% RSLogix 500 project PV8M.RSS, saved by version 8.30.00.16 %
PROJECT "PV8M"    % processor: Bul.1763 MicroLogix 1100 Series B %

PROGRAM FILES
  LAD 2   64 rungs

DATA FILES
  O0 OUTPUT  5 elements
  I1 INPUT  7 elements
  S2 STATUS  66 elements
  B3 BINARY  6 elements
  T4 TIMER  9 elements
  C5 COUNTER  1 elements
  R6 CONTROL  1 elements
  N7 INTEGER  11 elements
  F8 FLOAT  1 elements

LADDER 2
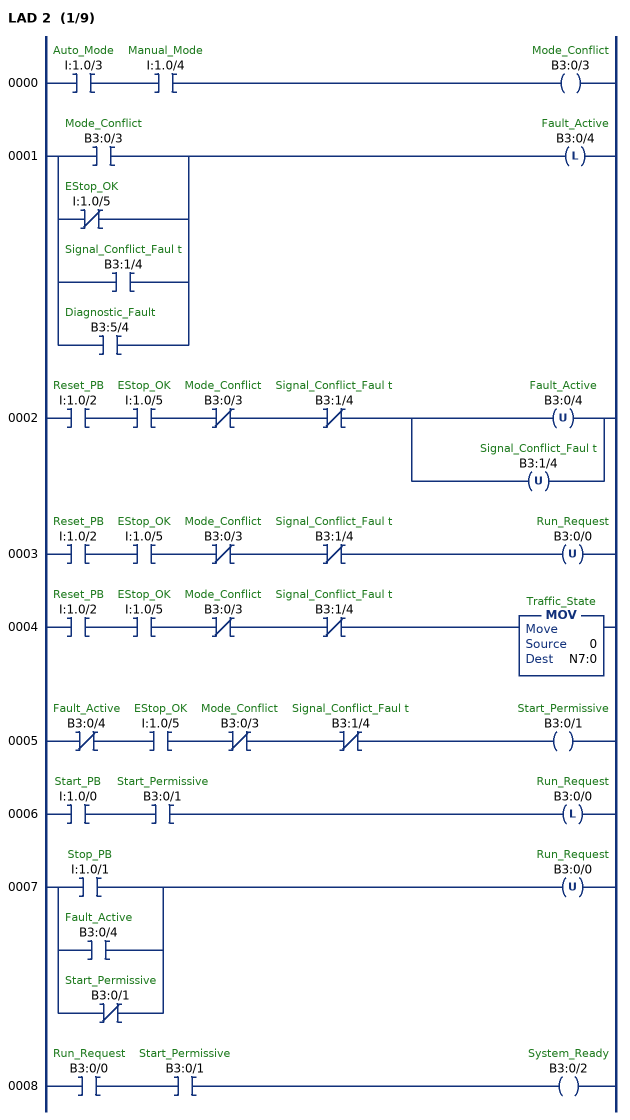
% Rung: 0 %
SOR XIC I:1.0/3 XIC I:1.0/4 OTE B3:0/3 EOR
%   I:1.0/3  "Auto_Mode" %
%   I:1.0/4  "Manual_Mode" %
%   B3:0/3  "Mode_Conflict" %
% Rung: 1 %
SOR BST XIC B3:0/3 NXB BST XIO I:1.0/5 NXB BST XIC B3:1/4 NXB XIC B3:5/4 BND BND BND OTL B3:0/4 EOR
%   B3:0/3  "Mode_Conflict" %
%   I:1.0/5  "EStop_OK" %
%   B3:1/4  "Signal_Conflict_Faul t" %
%   B3:5/4  "Diagnostic_Fault" %
%   B3:0/4  "Fault_Active" %
% Rung: 2 %
SOR XIC I:1.0/2 XIC I:1.0/5 XIO B3:0/3 XIO B3:1/4 BST OTU B3:0/4 NXB OTU B3:1/4 BND EOR
%   I:1.0/2  "Reset_PB" %
%   I:1.0/5  "EStop_OK" %
%   B3:0/3  "Mode_Conflict" %
%   B3:1/4  "Signal_Conflict_Faul t" %
%   B3:0/4  "Fault_Active" %
% Rung: 3 %
SOR XIC I:1.0/2 XIC I:1.0/5 XIO B3:0/3 XIO B3:1/4 OTU B3:0/0 EOR
%   I:1.0/2  "Reset_PB" %
%   I:1.0/5  "EStop_OK" %
%   B3:0/3  "Mode_Conflict" %
%   B3:1/4  "Signal_Conflict_Faul t" %
%   B3:0/0  "Run_Request" %
% Rung: 4 %
SOR XIC I:1.0/2 XIC I:1.0/5 XIO B3:0/3 XIO B3:1/4 MOV 0 N7:0 EOR
%   I:1.0/2  "Reset_PB" %
%   I:1.0/5  "EStop_OK" %
%   B3:0/3  "Mode_Conflict" %
%   B3:1/4  "Signal_Conflict_Faul t" %
%   N7:0  "Traffic_State" %
% Rung: 5 %
SOR XIO B3:0/4 XIC I:1.0/5 XIO B3:0/3 XIO B3:1/4 OTE B3:0/1 EOR
%   B3:0/4  "Fault_Active" %
%   I:1.0/5  "EStop_OK" %
%   B3:0/3  "Mode_Conflict" %
%   B3:1/4  "Signal_Conflict_Faul t" %
%   B3:0/1  "Start_Permissive" %
% Rung: 6 %
SOR XIC I:1.0/0 XIC B3:0/1 OTL B3:0/0 EOR
%   I:1.0/0  "Start_PB" %
%   B3:0/1  "Start_Permissive" %
%   B3:0/0  "Run_Request" %
% Rung: 7 %
SOR BST XIC I:1.0/1 NXB BST XIC B3:0/4 NXB XIO B3:0/1 BND BND OTU B3:0/0 EOR
%   I:1.0/1  "Stop_PB" %
%   B3:0/4  "Fault_Active" %
%   B3:0/1  "Start_Permissive" %
%   B3:0/0  "Run_Request" %
% Rung: 8 %
SOR XIC B3:0/0 XIC B3:0/1 OTE B3:0/2 EOR
%   B3:0/0  "Run_Request" %
%   B3:0/1  "Start_Permissive" %
%   B3:0/2  "System_Ready" %

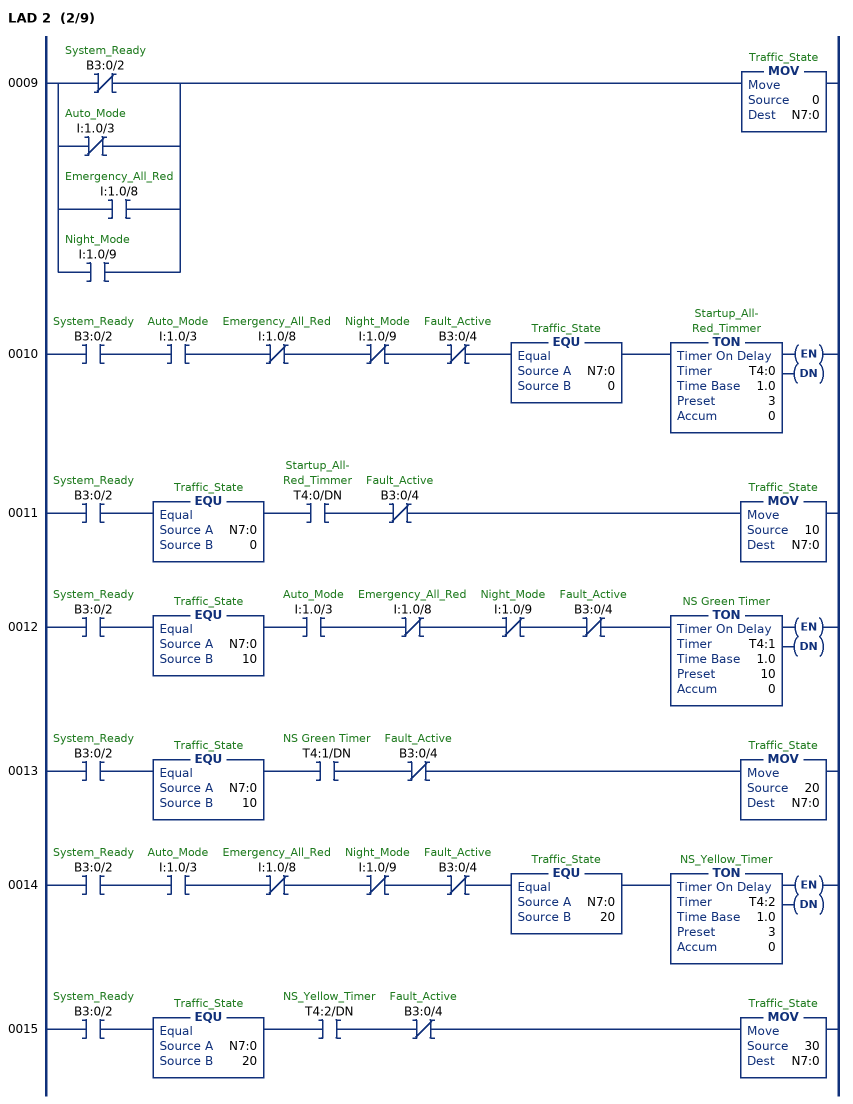
% Rung: 9 %
SOR BST XIO B3:0/2 NXB BST XIO I:1.0/3 NXB BST XIC I:1.0/8 NXB XIC I:1.0/9 BND BND BND MOV 0 N7:0 EOR
%   B3:0/2  "System_Ready" %
%   I:1.0/3  "Auto_Mode" %
%   I:1.0/8  "Emergency_All_Red" %
%   I:1.0/9  "Night_Mode" %
%   N7:0  "Traffic_State" %
% Rung: 10 %
SOR XIC B3:0/2 XIC I:1.0/3 XIO I:1.0/8 XIO I:1.0/9 XIO B3:0/4 EQU N7:0 0 TON T4:0 1.0 3 0 EOR
%   B3:0/2  "System_Ready" %
%   I:1.0/3  "Auto_Mode" %
%   I:1.0/8  "Emergency_All_Red" %
%   I:1.0/9  "Night_Mode" %
%   B3:0/4  "Fault_Active" %
%   N7:0  "Traffic_State" %
%   T4:0  "Startup_All- Red_Timmer" %
% Rung: 11 %
SOR XIC B3:0/2 EQU N7:0 0 XIC T4:0/DN XIO B3:0/4 MOV 10 N7:0 EOR
%   B3:0/2  "System_Ready" %
%   N7:0  "Traffic_State" %
%   T4:0  "Startup_All- Red_Timmer" %
%   B3:0/4  "Fault_Active" %
% Rung: 12 %
SOR XIC B3:0/2 EQU N7:0 10 XIC I:1.0/3 XIO I:1.0/8 XIO I:1.0/9 XIO B3:0/4 TON T4:1 1.0 10 0 EOR
%   B3:0/2  "System_Ready" %
%   N7:0  "Traffic_State" %
%   I:1.0/3  "Auto_Mode" %
%   I:1.0/8  "Emergency_All_Red" %
%   I:1.0/9  "Night_Mode" %
%   B3:0/4  "Fault_Active" %
%   T4:1  "NS Green Timer" %
% Rung: 13 %
SOR XIC B3:0/2 EQU N7:0 10 XIC T4:1/DN XIO B3:0/4 MOV 20 N7:0 EOR
%   B3:0/2  "System_Ready" %
%   N7:0  "Traffic_State" %
%   T4:1  "NS Green Timer" %
%   B3:0/4  "Fault_Active" %
% Rung: 14 %
SOR XIC B3:0/2 XIC I:1.0/3 XIO I:1.0/8 XIO I:1.0/9 XIO B3:0/4 EQU N7:0 20 TON T4:2 1.0 3 0 EOR
%   B3:0/2  "System_Ready" %
%   I:1.0/3  "Auto_Mode" %
%   I:1.0/8  "Emergency_All_Red" %
%   I:1.0/9  "Night_Mode" %
%   B3:0/4  "Fault_Active" %
%   N7:0  "Traffic_State" %
%   T4:2  "NS_Yellow_Timer" %
% Rung: 15 %
SOR XIC B3:0/2 EQU N7:0 20 XIC T4:2/DN XIO B3:0/4 MOV 30 N7:0 EOR
%   B3:0/2  "System_Ready" %
%   N7:0  "Traffic_State" %
%   T4:2  "NS_Yellow_Timer" %
%   B3:0/4  "Fault_Active" %

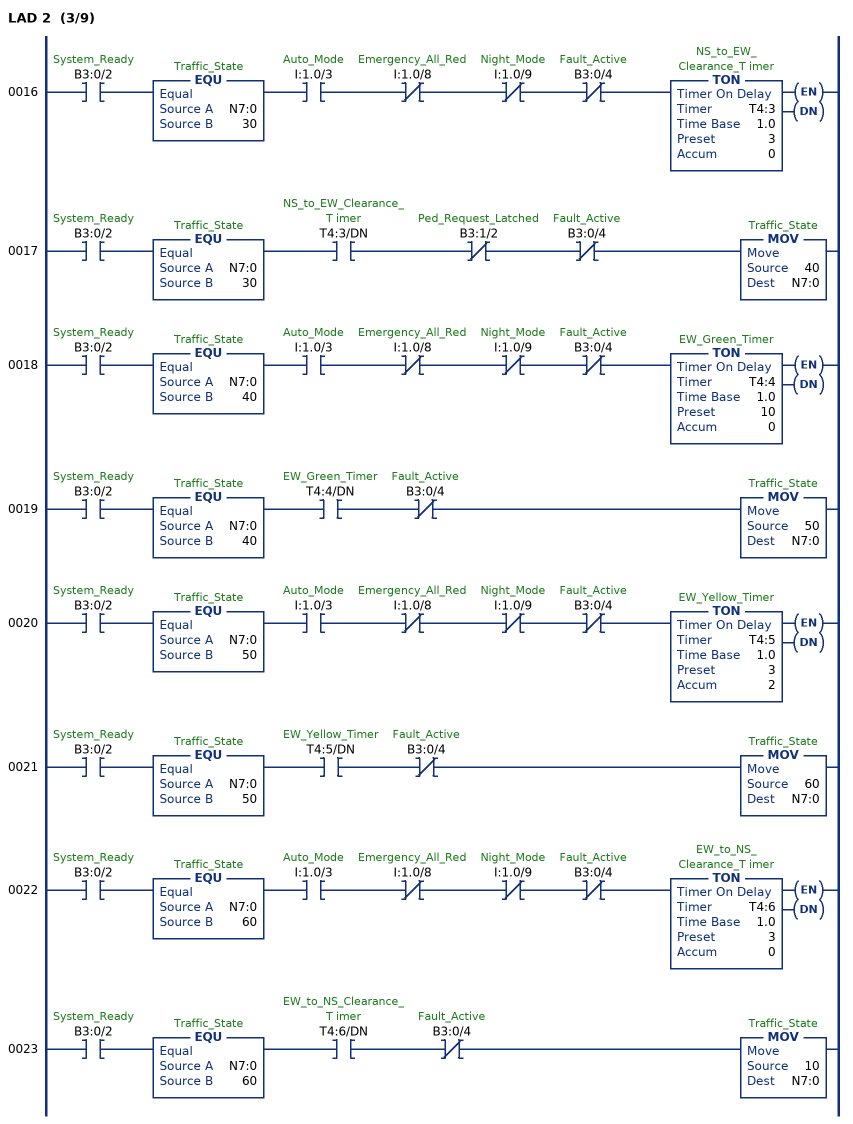
% Rung: 16 %
SOR XIC B3:0/2 EQU N7:0 30 XIC I:1.0/3 XIO I:1.0/8 XIO I:1.0/9 XIO B3:0/4 TON T4:3 1.0 3 0 EOR
%   B3:0/2  "System_Ready" %
%   N7:0  "Traffic_State" %
%   I:1.0/3  "Auto_Mode" %
%   I:1.0/8  "Emergency_All_Red" %
%   I:1.0/9  "Night_Mode" %
%   B3:0/4  "Fault_Active" %
%   T4:3  "NS_to_EW_Clearance_T imer" %
% Rung: 17 %
SOR XIC B3:0/2 EQU N7:0 30 XIC T4:3/DN XIO B3:1/2 XIO B3:0/4 MOV 40 N7:0 EOR
%   B3:0/2  "System_Ready" %
%   N7:0  "Traffic_State" %
%   T4:3  "NS_to_EW_Clearance_T imer" %
%   B3:1/2  "Ped_Request_Latched" %
%   B3:0/4  "Fault_Active" %
% Rung: 18 %
SOR XIC B3:0/2 EQU N7:0 40 XIC I:1.0/3 XIO I:1.0/8 XIO I:1.0/9 XIO B3:0/4 TON T4:4 1.0 10 0 EOR
%   B3:0/2  "System_Ready" %
%   N7:0  "Traffic_State" %
%   I:1.0/3  "Auto_Mode" %
%   I:1.0/8  "Emergency_All_Red" %
%   I:1.0/9  "Night_Mode" %
%   B3:0/4  "Fault_Active" %
%   T4:4  "EW_Green_Timer" %
% Rung: 19 %
SOR XIC B3:0/2 EQU N7:0 40 XIC T4:4/DN XIO B3:0/4 MOV 50 N7:0 EOR
%   B3:0/2  "System_Ready" %
%   N7:0  "Traffic_State" %
%   T4:4  "EW_Green_Timer" %
%   B3:0/4  "Fault_Active" %
% Rung: 20 %
SOR XIC B3:0/2 EQU N7:0 50 XIC I:1.0/3 XIO I:1.0/8 XIO I:1.0/9 XIO B3:0/4 TON T4:5 1.0 3 2 EOR
%   B3:0/2  "System_Ready" %
%   N7:0  "Traffic_State" %
%   I:1.0/3  "Auto_Mode" %
%   I:1.0/8  "Emergency_All_Red" %
%   I:1.0/9  "Night_Mode" %
%   B3:0/4  "Fault_Active" %
%   T4:5  "EW_Yellow_Timer" %
% Rung: 21 %
SOR XIC B3:0/2 EQU N7:0 50 XIC T4:5/DN XIO B3:0/4 MOV 60 N7:0 EOR
%   B3:0/2  "System_Ready" %
%   N7:0  "Traffic_State" %
%   T4:5  "EW_Yellow_Timer" %
%   B3:0/4  "Fault_Active" %
% Rung: 22 %
SOR XIC B3:0/2 EQU N7:0 60 XIC I:1.0/3 XIO I:1.0/8 XIO I:1.0/9 XIO B3:0/4 TON T4:6 1.0 3 0 EOR
%   B3:0/2  "System_Ready" %
%   N7:0  "Traffic_State" %
%   I:1.0/3  "Auto_Mode" %
%   I:1.0/8  "Emergency_All_Red" %
%   I:1.0/9  "Night_Mode" %
%   B3:0/4  "Fault_Active" %
%   T4:6  "EW_to_NS_Clearance_T imer" %
% Rung: 23 %
SOR XIC B3:0/2 EQU N7:0 60 XIC T4:6/DN XIO B3:0/4 MOV 10 N7:0 EOR
%   B3:0/2  "System_Ready" %
%   N7:0  "Traffic_State" %
%   T4:6  "EW_to_NS_Clearance_T imer" %
%   B3:0/4  "Fault_Active" %

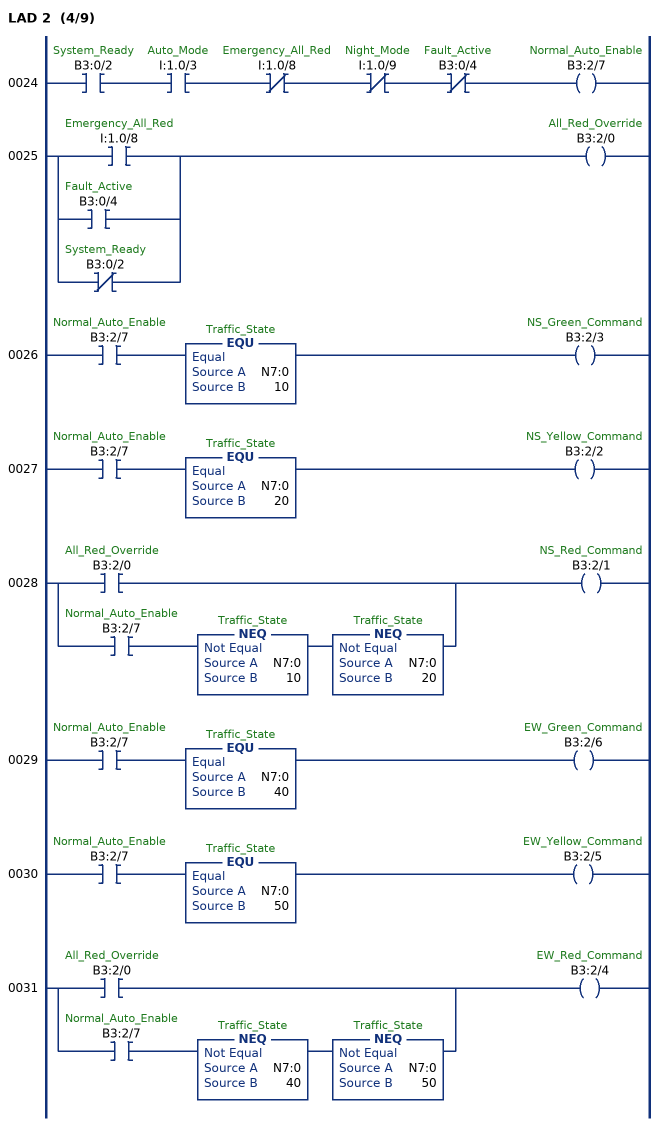
% Rung: 24 %
SOR XIC B3:0/2 XIC I:1.0/3 XIO I:1.0/8 XIO I:1.0/9 XIO B3:0/4 OTE B3:2/7 EOR
%   B3:0/2  "System_Ready" %
%   I:1.0/3  "Auto_Mode" %
%   I:1.0/8  "Emergency_All_Red" %
%   I:1.0/9  "Night_Mode" %
%   B3:0/4  "Fault_Active" %
%   B3:2/7  "Normal_Auto_Enable" %
% Rung: 25 %
SOR BST XIC I:1.0/8 NXB BST XIC B3:0/4 NXB XIO B3:0/2 BND BND OTE B3:2/0 EOR
%   I:1.0/8  "Emergency_All_Red" %
%   B3:0/4  "Fault_Active" %
%   B3:0/2  "System_Ready" %
%   B3:2/0  "All_Red_Override" %
% Rung: 26 %
SOR XIC B3:2/7 EQU N7:0 10 OTE B3:2/3 EOR
%   B3:2/7  "Normal_Auto_Enable" %
%   N7:0  "Traffic_State" %
%   B3:2/3  "NS_Green_Command" %
% Rung: 27 %
SOR XIC B3:2/7 EQU N7:0 20 OTE B3:2/2 EOR
%   B3:2/7  "Normal_Auto_Enable" %
%   N7:0  "Traffic_State" %
%   B3:2/2  "NS_Yellow_Command" %
% Rung: 28 %
SOR BST XIC B3:2/0 NXB XIC B3:2/7 NEQ N7:0 10 NEQ N7:0 20 BND OTE B3:2/1 EOR
%   B3:2/0  "All_Red_Override" %
%   B3:2/7  "Normal_Auto_Enable" %
%   N7:0  "Traffic_State" %
%   B3:2/1  "NS_Red_Command" %
% Rung: 29 %
SOR XIC B3:2/7 EQU N7:0 40 OTE B3:2/6 EOR
%   B3:2/7  "Normal_Auto_Enable" %
%   N7:0  "Traffic_State" %
%   B3:2/6  "EW_Green_Command" %
% Rung: 30 %
SOR XIC B3:2/7 EQU N7:0 50 OTE B3:2/5 EOR
%   B3:2/7  "Normal_Auto_Enable" %
%   N7:0  "Traffic_State" %
%   B3:2/5  "EW_Yellow_Command" %
% Rung: 31 %
SOR BST XIC B3:2/0 NXB XIC B3:2/7 NEQ N7:0 40 NEQ N7:0 50 BND OTE B3:2/4 EOR
%   B3:2/0  "All_Red_Override" %
%   B3:2/7  "Normal_Auto_Enable" %
%   N7:0  "Traffic_State" %
%   B3:2/4  "EW_Red_Command" %

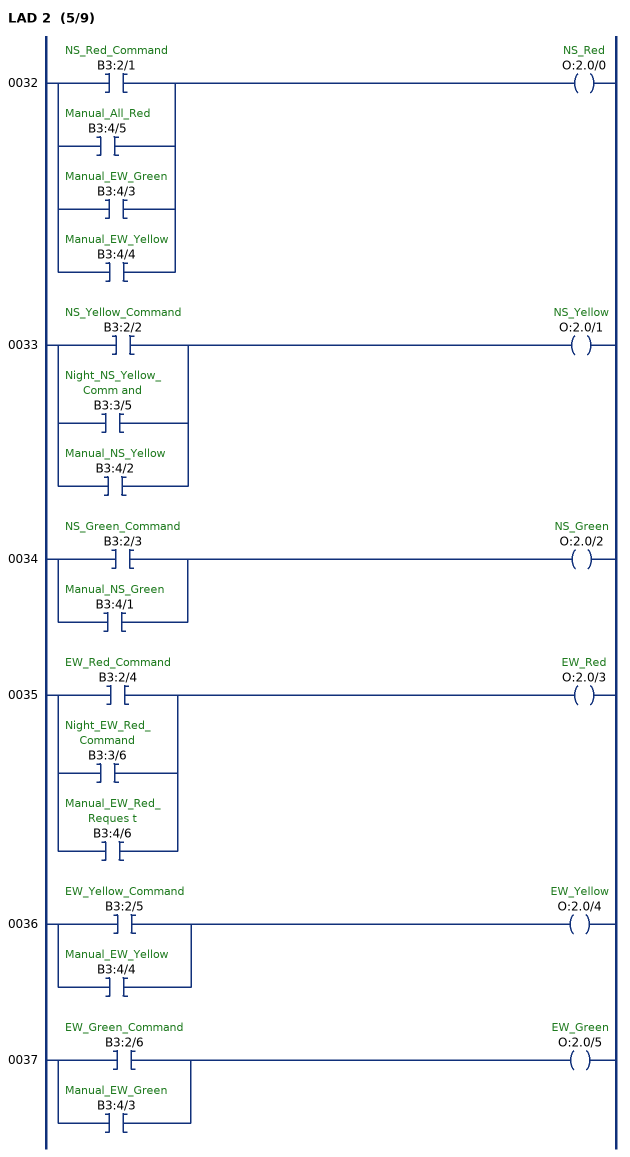
% Rung: 32 %
SOR BST XIC B3:2/1 NXB BST XIC B3:4/5 NXB BST XIC B3:4/3 NXB XIC B3:4/4 BND BND BND OTE O:2.0/0 EOR
%   B3:2/1  "NS_Red_Command" %
%   B3:4/5  "Manual_All_Red" %
%   B3:4/3  "Manual_EW_Green" %
%   B3:4/4  "Manual_EW_Yellow" %
%   O:2.0/0  "NS_Red" %
% Rung: 33 %
SOR BST XIC B3:2/2 NXB BST XIC B3:3/5 NXB XIC B3:4/2 BND BND OTE O:2.0/1 EOR
%   B3:2/2  "NS_Yellow_Command" %
%   B3:3/5  "Night_NS_Yellow_Comm and" %
%   B3:4/2  "Manual_NS_Yellow" %
%   O:2.0/1  "NS_Yellow" %
% Rung: 34 %
SOR BST XIC B3:2/3 NXB XIC B3:4/1 BND OTE O:2.0/2 EOR
%   B3:2/3  "NS_Green_Command" %
%   B3:4/1  "Manual_NS_Green" %
%   O:2.0/2  "NS_Green" %
% Rung: 35 %
SOR BST XIC B3:2/4 NXB BST XIC B3:3/6 NXB XIC B3:4/6 BND BND OTE O:2.0/3 EOR
%   B3:2/4  "EW_Red_Command" %
%   B3:3/6  "Night_EW_Red_Command" %
%   B3:4/6  "Manual_EW_Red_Reques t" %
%   O:2.0/3  "EW_Red" %
% Rung: 36 %
SOR BST XIC B3:2/5 NXB XIC B3:4/4 BND OTE O:2.0/4 EOR
%   B3:2/5  "EW_Yellow_Command" %
%   B3:4/4  "Manual_EW_Yellow" %
%   O:2.0/4  "EW_Yellow" %
% Rung: 37 %
SOR BST XIC B3:2/6 NXB XIC B3:4/3 BND OTE O:2.0/5 EOR
%   B3:2/6  "EW_Green_Command" %
%   B3:4/3  "Manual_EW_Green" %
%   O:2.0/5  "EW_Green" %

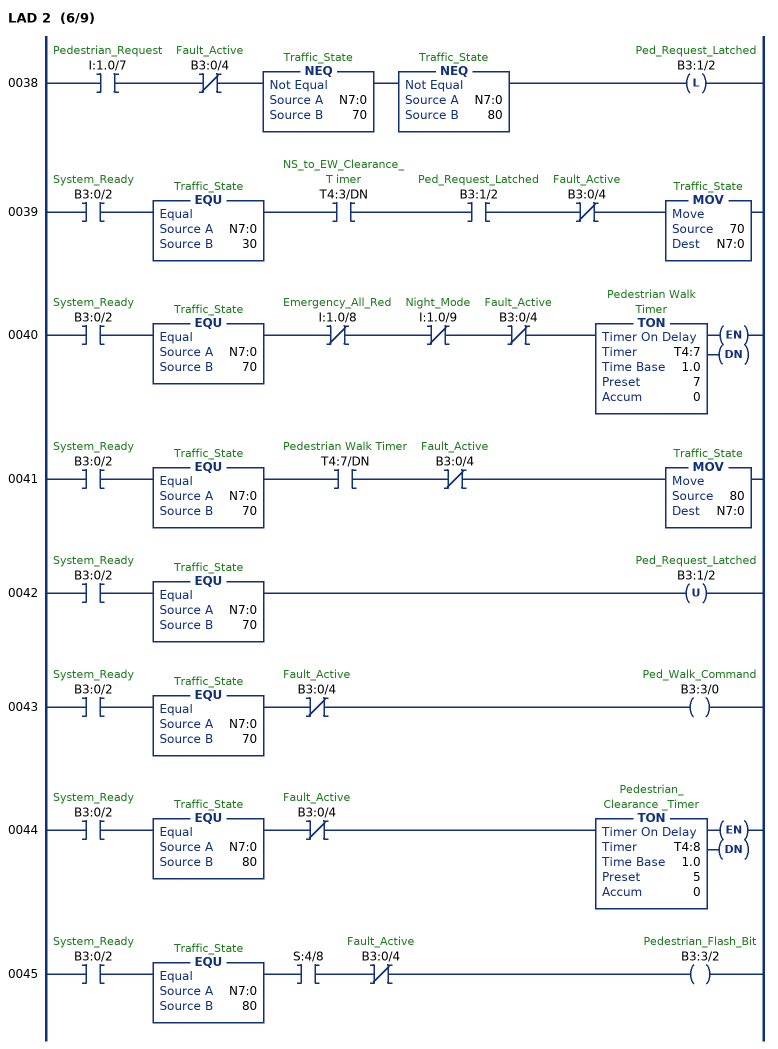
% Rung: 38 %
SOR XIC I:1.0/7 XIO B3:0/4 NEQ N7:0 70 NEQ N7:0 80 OTL B3:1/2 EOR
%   I:1.0/7  "Pedestrian_Request" %
%   B3:0/4  "Fault_Active" %
%   N7:0  "Traffic_State" %
%   B3:1/2  "Ped_Request_Latched" %
% Rung: 39 %
SOR XIC B3:0/2 EQU N7:0 30 XIC T4:3/DN XIC B3:1/2 XIO B3:0/4 MOV 70 N7:0 EOR
%   B3:0/2  "System_Ready" %
%   N7:0  "Traffic_State" %
%   T4:3  "NS_to_EW_Clearance_T imer" %
%   B3:1/2  "Ped_Request_Latched" %
%   B3:0/4  "Fault_Active" %
% Rung: 40 %
SOR XIC B3:0/2 EQU N7:0 70 XIO I:1.0/8 XIO I:1.0/9 XIO B3:0/4 TON T4:7 1.0 7 0 EOR
%   B3:0/2  "System_Ready" %
%   N7:0  "Traffic_State" %
%   I:1.0/8  "Emergency_All_Red" %
%   I:1.0/9  "Night_Mode" %
%   B3:0/4  "Fault_Active" %
%   T4:7  "Pedestrian Walk Timer" %
% Rung: 41 %
SOR XIC B3:0/2 EQU N7:0 70 XIC T4:7/DN XIO B3:0/4 MOV 80 N7:0 EOR
%   B3:0/2  "System_Ready" %
%   N7:0  "Traffic_State" %
%   T4:7  "Pedestrian Walk Timer" %
%   B3:0/4  "Fault_Active" %
% Rung: 42 %
SOR XIC B3:0/2 EQU N7:0 70 OTU B3:1/2 EOR
%   B3:0/2  "System_Ready" %
%   N7:0  "Traffic_State" %
%   B3:1/2  "Ped_Request_Latched" %
% Rung: 43 %
SOR XIC B3:0/2 EQU N7:0 70 XIO B3:0/4 OTE B3:3/0 EOR
%   B3:0/2  "System_Ready" %
%   N7:0  "Traffic_State" %
%   B3:0/4  "Fault_Active" %
%   B3:3/0  "Ped_Walk_Command" %
% Rung: 44 %
SOR XIC B3:0/2 EQU N7:0 80 XIO B3:0/4 TON T4:8 1.0 5 0 EOR
%   B3:0/2  "System_Ready" %
%   N7:0  "Traffic_State" %
%   B3:0/4  "Fault_Active" %
%   T4:8  "Pedestrian_Clearance _Timer" %
% Rung: 45 %
SOR XIC B3:0/2 EQU N7:0 80 XIC S:4/8 XIO B3:0/4 OTE B3:3/2 EOR
%   B3:0/2  "System_Ready" %
%   N7:0  "Traffic_State" %
%   B3:0/4  "Fault_Active" %
%   B3:3/2  "Pedestrian_Flash_Bit" %

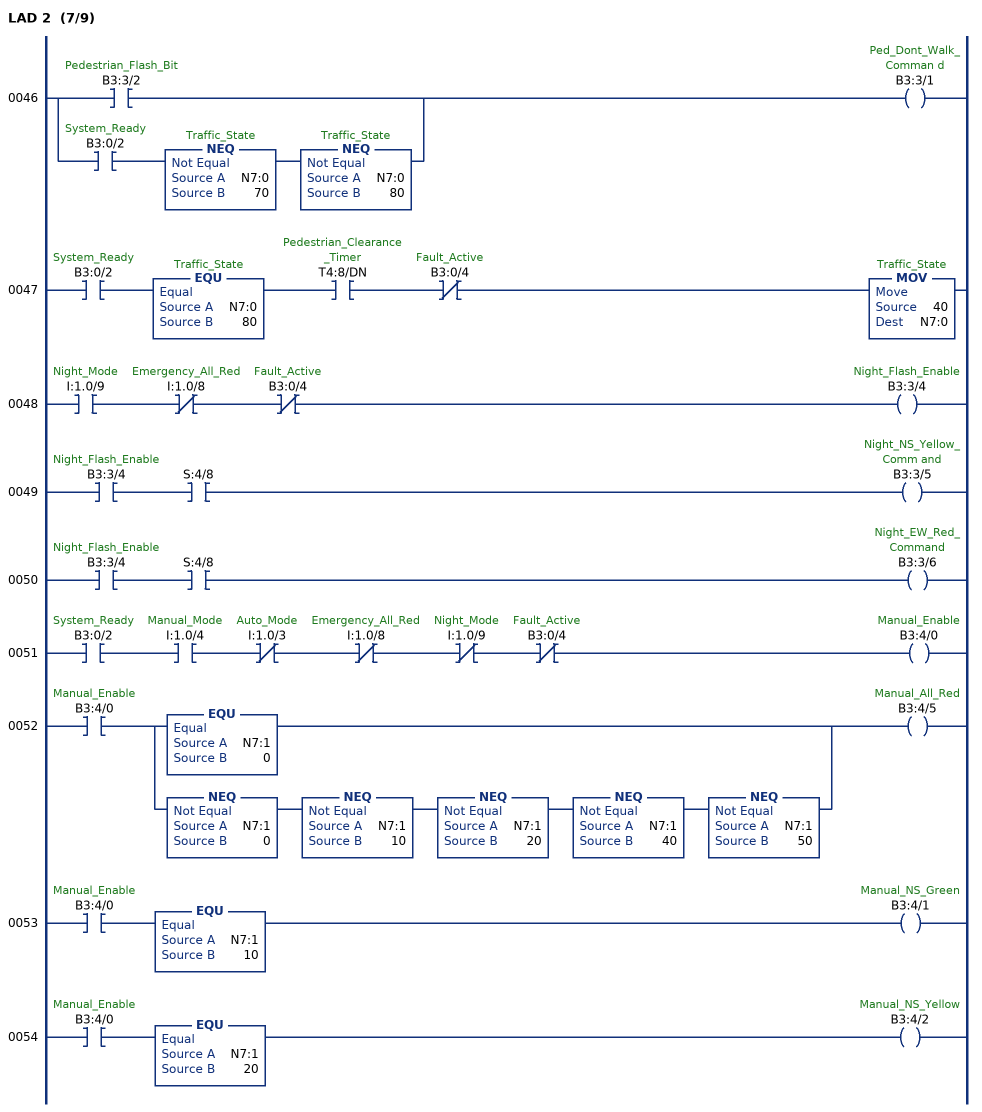
% Rung: 46 %
SOR BST XIC B3:3/2 NXB XIC B3:0/2 NEQ N7:0 70 NEQ N7:0 80 BND OTE B3:3/1 EOR
%   B3:3/2  "Pedestrian_Flash_Bit" %
%   B3:0/2  "System_Ready" %
%   N7:0  "Traffic_State" %
%   B3:3/1  "Ped_Dont_Walk_Comman d" %
% Rung: 47 %
SOR XIC B3:0/2 EQU N7:0 80 XIC T4:8/DN XIO B3:0/4 MOV 40 N7:0 EOR
%   B3:0/2  "System_Ready" %
%   N7:0  "Traffic_State" %
%   T4:8  "Pedestrian_Clearance _Timer" %
%   B3:0/4  "Fault_Active" %
% Rung: 48 %
SOR XIC I:1.0/9 XIO I:1.0/8 XIO B3:0/4 OTE B3:3/4 EOR
%   I:1.0/9  "Night_Mode" %
%   I:1.0/8  "Emergency_All_Red" %
%   B3:0/4  "Fault_Active" %
%   B3:3/4  "Night_Flash_Enable" %
% Rung: 49 %
SOR XIC B3:3/4 XIC S:4/8 OTE B3:3/5 EOR
%   B3:3/4  "Night_Flash_Enable" %
%   B3:3/5  "Night_NS_Yellow_Comm and" %
% Rung: 50 %
SOR XIC B3:3/4 XIC S:4/8 OTE B3:3/6 EOR
%   B3:3/4  "Night_Flash_Enable" %
%   B3:3/6  "Night_EW_Red_Command" %
% Rung: 51 %
SOR XIC B3:0/2 XIC I:1.0/4 XIO I:1.0/3 XIO I:1.0/8 XIO I:1.0/9 XIO B3:0/4 OTE B3:4/0 EOR
%   B3:0/2  "System_Ready" %
%   I:1.0/4  "Manual_Mode" %
%   I:1.0/3  "Auto_Mode" %
%   I:1.0/8  "Emergency_All_Red" %
%   I:1.0/9  "Night_Mode" %
%   B3:0/4  "Fault_Active" %
%   B3:4/0  "Manual_Enable" %
% Rung: 52 %
SOR XIC B3:4/0 BST EQU N7:1 0 NXB NEQ N7:1 0 NEQ N7:1 10 NEQ N7:1 20 NEQ N7:1 40 NEQ N7:1 50 BND OTE B3:4/5 EOR
%   B3:4/0  "Manual_Enable" %
%   B3:4/5  "Manual_All_Red" %
% Rung: 53 %
SOR XIC B3:4/0 EQU N7:1 10 OTE B3:4/1 EOR
%   B3:4/0  "Manual_Enable" %
%   B3:4/1  "Manual_NS_Green" %
% Rung: 54 %
SOR XIC B3:4/0 EQU N7:1 20 OTE B3:4/2 EOR
%   B3:4/0  "Manual_Enable" %
%   B3:4/2  "Manual_NS_Yellow" %

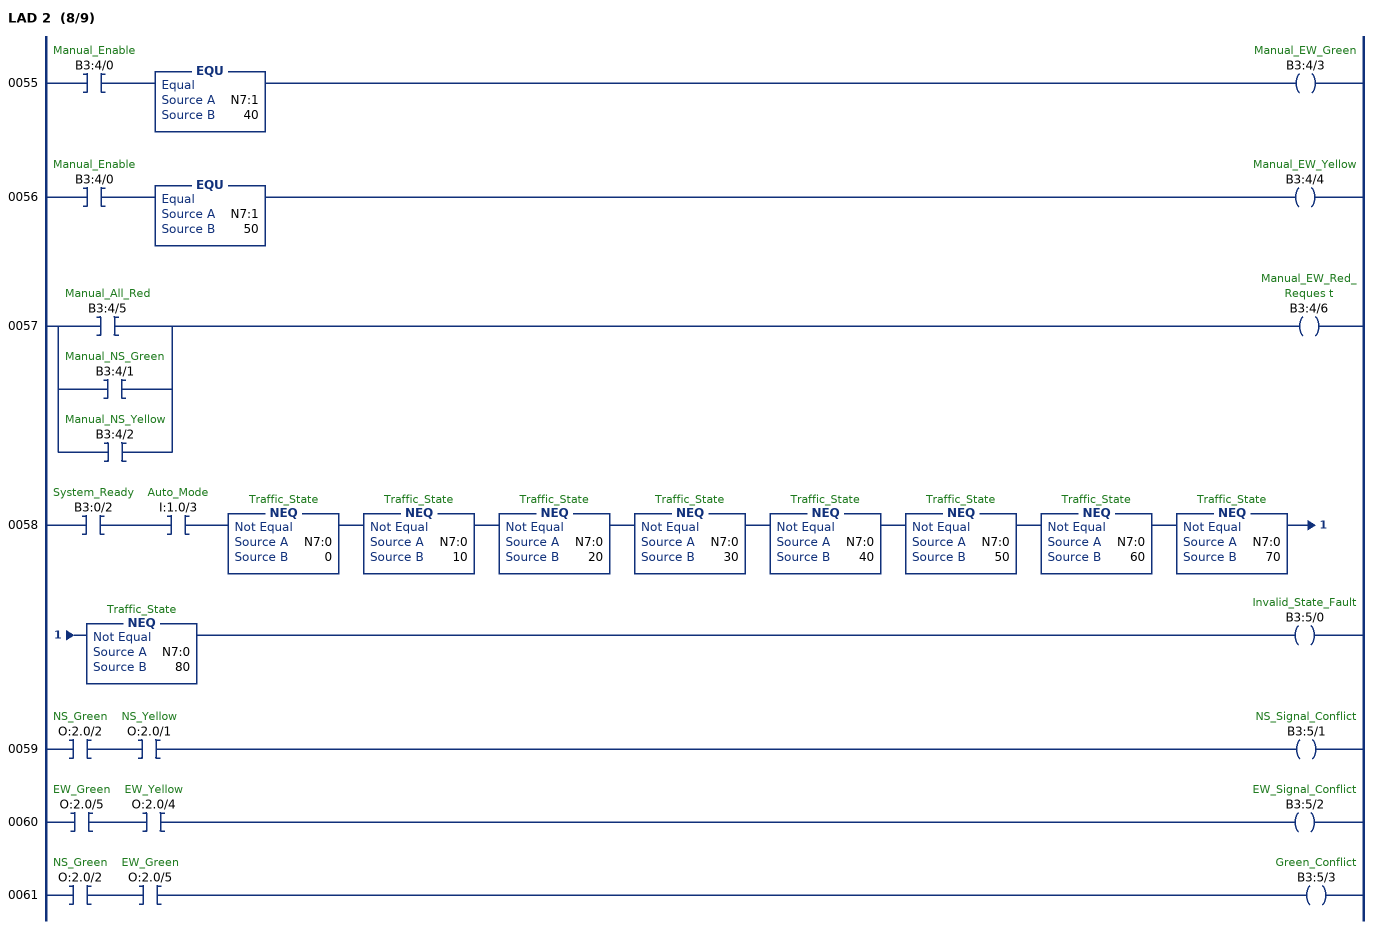
% Rung: 55 %
SOR XIC B3:4/0 EQU N7:1 40 OTE B3:4/3 EOR
%   B3:4/0  "Manual_Enable" %
%   B3:4/3  "Manual_EW_Green" %
% Rung: 56 %
SOR XIC B3:4/0 EQU N7:1 50 OTE B3:4/4 EOR
%   B3:4/0  "Manual_Enable" %
%   B3:4/4  "Manual_EW_Yellow" %
% Rung: 57 %
SOR BST XIC B3:4/5 NXB BST XIC B3:4/1 NXB XIC B3:4/2 BND BND OTE B3:4/6 EOR
%   B3:4/5  "Manual_All_Red" %
%   B3:4/1  "Manual_NS_Green" %
%   B3:4/2  "Manual_NS_Yellow" %
%   B3:4/6  "Manual_EW_Red_Reques t" %
% Rung: 58 %
SOR XIC B3:0/2 XIC I:1.0/3 NEQ N7:0 0 NEQ N7:0 10 NEQ N7:0 20 NEQ N7:0 30 NEQ N7:0 40 NEQ N7:0 50 NEQ N7:0 60 NEQ N7:0 70 NEQ N7:0 80 OTE B3:5/0 EOR
%   B3:0/2  "System_Ready" %
%   I:1.0/3  "Auto_Mode" %
%   N7:0  "Traffic_State" %
%   B3:5/0  "Invalid_State_Fault" %
% Rung: 59 %
SOR XIC O:2.0/2 XIC O:2.0/1 OTE B3:5/1 EOR
%   O:2.0/2  "NS_Green" %
%   O:2.0/1  "NS_Yellow" %
%   B3:5/1  "NS_Signal_Conflict" %
% Rung: 60 %
SOR XIC O:2.0/5 XIC O:2.0/4 OTE B3:5/2 EOR
%   O:2.0/5  "EW_Green" %
%   O:2.0/4  "EW_Yellow" %
%   B3:5/2  "EW_Signal_Conflict" %
% Rung: 61 %
SOR XIC O:2.0/2 XIC O:2.0/5 OTE B3:5/3 EOR
%   O:2.0/2  "NS_Green" %
%   O:2.0/5  "EW_Green" %
%   B3:5/3  "Green_Conflict" %

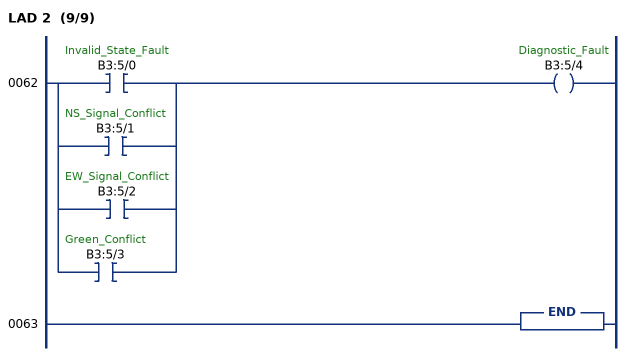
% Rung: 62 %
SOR BST XIC B3:5/0 NXB BST XIC B3:5/1 NXB BST XIC B3:5/2 NXB XIC B3:5/3 BND BND BND OTE B3:5/4 EOR
%   B3:5/0  "Invalid_State_Fault" %
%   B3:5/1  "NS_Signal_Conflict" %
%   B3:5/2  "EW_Signal_Conflict" %
%   B3:5/3  "Green_Conflict" %
%   B3:5/4  "Diagnostic_Fault" %
% Rung: 63 %
SOR END EOR

OTHER DOCUMENTED ADDRESSES
  B3:0/5  "ALL_Red_Step"
  B3:0/6  "NS_Green_Step"
  B3:0/7  "NS_Yellow_Step"
  B3:1/0  "EW_Green_Step"
  B3:1/1  "EW_Yellow_Step"
  B3:1/5  "Next_EW_Direction"
  B3:3/3  "Ped_DontWalk_Steady"
  I:1.0/6  "Signal_Conflict_Faul t"
  N7  

DATA TABLE (non-zero values as saved)
DATA B3
% B3:0 % 0X0007 0X0000 0X00A2 0X0002 0X0000 0X0000
DATA T4
% .PRE .ACC %
% T4:0 % 3 0
% T4:1 % 10 0
% T4:2 % 3 0
% T4:3 % 3 0
% T4:4 % 10 0
% T4:5 % 3 2
% T4:6 % 3 0
% T4:7 % 7 0
% T4:8 % 5 0
DATA N7
% N7:0 % 50 35 0 0 0 0 0 0 0 0
% N7:10 % 30
